FUNCTION_BLOCK FB_ModuleReferenceBindingContext IMPLEMENTS I_ModuleReferenceBindings
VAR_OUTPUT
	Error : BOOL;
	ErrorMessage : STRING(255);
END_VAR
VAR
	_Names : ARRAY[1..Param_Config.MaxModuleReferences] OF STRING(80);
	_SourceNames : ARRAY[1..Param_Config.MaxModuleReferences] OF STRING(255);
	_Consumed : ARRAY[1..Param_Config.MaxModuleReferences] OF BOOL;
	_ReferenceManager : REFERENCE TO FB_ReferenceManager;
	_Count : UINT;
	_Active : BOOL;
END_VAR

METHOD PUBLIC M_Begin : BOOL
VAR_IN_OUT CONSTANT
	ModuleConfig : ST_ModuleFileConfig;
END_VAR
VAR_IN_OUT
	ReferenceManager : FB_ReferenceManager;
END_VAR
VAR
	nItem : UINT;
	nOther : UINT;
END_VAR
M_Begin := FALSE;
M_Clear();

IF ModuleConfig.ReferenceCount > Param_Config.MaxModuleReferences THEN
	Error := TRUE;
	ErrorMessage := 'Module reference capacity was exceeded.';
	RETURN;
END_IF

FOR nItem := 1 TO ModuleConfig.ReferenceCount DO
	IF (ModuleConfig.References[nItem].Name = '') OR (ModuleConfig.References[nItem].Source = '') THEN
		Error := TRUE;
		ErrorMessage := 'Every Module reference requires a name and source.';
		RETURN;
	END_IF

	IF nItem > 1 THEN
		FOR nOther := 1 TO nItem - 1 DO
			IF ModuleConfig.References[nOther].Name = ModuleConfig.References[nItem].Name THEN
				Error := TRUE;
				ErrorMessage := CONCAT('Duplicate Module reference name: ', ModuleConfig.References[nItem].Name);
				RETURN;
			END_IF
		END_FOR
	END_IF

	_Names[nItem] := ModuleConfig.References[nItem].Name;
	_SourceNames[nItem] := ModuleConfig.References[nItem].Source;
END_FOR

_Count := ModuleConfig.ReferenceCount;
_ReferenceManager REF= ReferenceManager;
_Active := TRUE;
M_Begin := TRUE;
END_METHOD

METHOD PUBLIC M_Clear
VAR
	nItem : UINT;
END_VAR
FOR nItem := 1 TO Param_Config.MaxModuleReferences DO
	_Names[nItem] := '';
	_SourceNames[nItem] := '';
	_Consumed[nItem] := FALSE;
END_FOR
_Count := 0;
_Active := FALSE;
Error := FALSE;
ErrorMessage := '';
END_METHOD

METHOD PUBLIC M_End : BOOL
VAR
	nItem : UINT;
END_VAR
M_End := FALSE;
IF Error THEN
	RETURN;
END_IF
IF NOT _Active THEN
	Error := TRUE;
	ErrorMessage := 'No Module reference binding context is active.';
	RETURN;
END_IF

FOR nItem := 1 TO _Count DO
	IF NOT _Consumed[nItem] THEN
		Error := TRUE;
		ErrorMessage := CONCAT('Unknown Module reference name: ', _Names[nItem]);
		RETURN;
	END_IF
END_FOR

_Active := FALSE;
M_End := TRUE;
END_METHOD

METHOD PRIVATE M_Take : I_BaseUnit
VAR_INPUT
	Name : STRING(80);
	Required : BOOL;
END_VAR
VAR_OUTPUT
	Present : BOOL;
	TakeErrorMessage : STRING(255);
END_VAR
VAR
	nItem : UINT;
	BaseUnit : I_BaseUnit;
END_VAR
M_Take := 0;
Present := FALSE;
TakeErrorMessage := '';
IF Error THEN
	TakeErrorMessage := ErrorMessage;
	RETURN;
END_IF
IF NOT _Active THEN
	Error := TRUE;
	ErrorMessage := 'No Module reference binding context is active.';
	TakeErrorMessage := ErrorMessage;
	RETURN;
END_IF
IF Name = '' THEN
	Error := TRUE;
	ErrorMessage := 'A Module reference name is required.';
	TakeErrorMessage := ErrorMessage;
	RETURN;
END_IF

FOR nItem := 1 TO _Count DO
	IF _Names[nItem] = Name THEN
		IF _Consumed[nItem] THEN
			Error := TRUE;
			ErrorMessage := CONCAT('Module reference was taken more than once: ', Name);
			TakeErrorMessage := ErrorMessage;
			RETURN;
		END_IF
		IF NOT __ISVALIDREF(_ReferenceManager) THEN
			Error := TRUE;
			ErrorMessage := 'The Module reference source registry is unavailable.';
			TakeErrorMessage := ErrorMessage;
			RETURN;
		END_IF
		BaseUnit := _ReferenceManager.M_Resolve(Name := _SourceNames[nItem]);
		IF BaseUnit = 0 THEN
			Error := TRUE;
			ErrorMessage := CONCAT('Module reference source was not registered: ', _SourceNames[nItem]);
			TakeErrorMessage := ErrorMessage;
			RETURN;
		END_IF
		_Consumed[nItem] := TRUE;
		Present := TRUE;
		M_Take := BaseUnit;
		RETURN;
	END_IF
END_FOR

IF Required THEN
	Error := TRUE;
	ErrorMessage := CONCAT('Missing required Module reference: ', Name);
	TakeErrorMessage := ErrorMessage;
END_IF
END_METHOD

METHOD PUBLIC M_TakeOptional : I_BaseUnit
VAR_INPUT
	Name : STRING(80);
END_VAR
VAR_OUTPUT
	Present : BOOL;
	ErrorMessage : STRING(255);
END_VAR
M_TakeOptional := M_Take(
	Name := Name,
	Required := FALSE,
	Present => Present,
	TakeErrorMessage => ErrorMessage);
END_METHOD

METHOD PUBLIC M_TakeRequired : I_BaseUnit
VAR_INPUT
	Name : STRING(80);
END_VAR
VAR_OUTPUT
	ErrorMessage : STRING(255);
END_VAR
VAR
	bPresent : BOOL;
END_VAR
M_TakeRequired := M_Take(
	Name := Name,
	Required := TRUE,
	Present => bPresent,
	TakeErrorMessage => ErrorMessage);
END_METHOD

END_FUNCTION_BLOCK

(* stored: Version 1.1.0.1, ProductVersion 3.1.4026.18
   POU FB_ModuleReferenceBindingContext: Id {7c687abe-a516-4907-99a9-0661f4a113f7}, SpecialFunc None
   Method M_Begin: Id {d1d908f7-7116-4aa5-bd31-ad596ff3d464}
   Method M_Clear: Id {9f5ed9e6-782a-49ae-8810-42d8923535b7}
   Method M_End: Id {e65b0cba-cfb5-4d8f-a0c3-e59ec5e5f652}
   Method M_Take: Id {19807c50-ad7f-4d30-8dae-3aa0f1f66969}
   Method M_TakeOptional: Id {c3a09870-d30e-44d5-a044-51ed5d29616d}
   Method M_TakeRequired: Id {d27284f7-cb21-485f-b2b5-2ebde4f660fc} *)
